(* IEC 61131-3 sources: cc_kush_rewrite/Functions/Bunker, 10 files *)

(* ---- FC_Bunker_CheckCriticalWeight.st ---- *)
FUNCTION FC_Bunker_CheckCriticalWeight : BOOL
VAR_INPUT
	Bunker1 : REFERENCE TO ST_Bunker;
	Bunker2 : REFERENCE TO ST_Bunker;
	Bunker3 : REFERENCE TO ST_Bunker;
END_VAR
VAR
END_VAR
// ========================================
// ПРОВЕРКА КРИТИЧЕСКИ НИЗКОГО ВЕСА
// ========================================
// Функция возвращает TRUE, если хотя бы один из бункеров достиг
// критически низкого уровня веса (сырье закончилось)
//
// ЛОГИКА:
// Когда определенное сырье заканчивается, вес бункера становится
// критически низким (rWeight <= BUNKER_WEIGHT_LIGHT_RED_SPECIAL).
// В этом случае необходимо подать красный сигнал на ВСЕ 3 бункера,
// чтобы прекратить подачу остального сырья. Далее они спокойно
// опустошаются в обычном автоматическом режиме.

FC_Bunker_CheckCriticalWeight :=
	(Bunker1.rWeight <= BUNKER_WEIGHT_LIGHT_RED_SPECIAL)
	OR (Bunker2.rWeight <= BUNKER_WEIGHT_LIGHT_RED_SPECIAL)
	OR (Bunker3.rWeight <= BUNKER_WEIGHT_LIGHT_RED_SPECIAL);

END_FUNCTION

(* ---- FC_Bunker_CheckEmptyBunker.st ---- *)
FUNCTION FC_Bunker_CheckEmptyBunker : BOOL
VAR_INPUT
	Bunker1 : REFERENCE TO ST_Bunker;
	Bunker2 : REFERENCE TO ST_Bunker;
	Bunker3 : REFERENCE TO ST_Bunker;
END_VAR
VAR
END_VAR
// ========================================
// ПРОВЕРКА ПОЛНОГО ОПУСТОШЕНИЯ БУНКЕРОВ
// ========================================
// Функция возвращает TRUE, если хотя бы один из бункеров полностью пуст.
//
// ЛОГИКА:
// Как только один из бункеров становится пустым (rWeight <= BUNKER_MINIMAL_WEIGHT),
// необходимо сразу остановить ВСЕ бункеры. Конвейер и отвалообразователь
// продолжают свою работу для транспортировки оставшегося материала.

FC_Bunker_CheckEmptyBunker :=
	(Bunker1.rWeight <= BUNKER_MINIMAL_WEIGHT)
	OR (Bunker2.rWeight <= BUNKER_MINIMAL_WEIGHT)
	OR (Bunker3.rWeight <= BUNKER_MINIMAL_WEIGHT);

END_FUNCTION

(* ---- FC_Bunker_CheckWeight.st ---- *)
FUNCTION FC_Bunker_CheckWeight : BOOL
VAR_INPUT
	Bunker : REFERENCE TO ST_Bunker;
END_VAR
VAR
END_VAR
// Проверка веса бункера. True - вес в порядке
FC_Bunker_CheckWeight := Bunker.rWeight > BUNKER_MINIMAL_WEIGHT;

END_FUNCTION

(* ---- FC_Bunker_EmergencyStop.st ---- *)
FUNCTION FC_Bunker_EmergencyStop : BOOL
VAR_INPUT
	Bunker : ST_Bunker;
END_VAR
VAR
	j : INT;
END_VAR
// Остановка моторов вибраторов (4 шт на бункер)
FOR j := 1 TO 4 DO
	Bunker.MotorVibrator[j].qxKM_Power := FALSE;
	Bunker.MotorVibrator[j].VFD.qxStart := FALSE;
	Bunker.MotorVibrator[j].VFD.Frequency.rTargetFrequency := 0.0;
	Bunker.MotorVibrator[j].VFD.qrOutFrequency := 0.0;
END_FOR

// Остановка моторов вибропитателей (2 шт на бункер)
FOR j := 1 TO 2 DO
	Bunker.MotorVibFeeder[j].qxKM_Power := FALSE;
	Bunker.MotorVibFeeder[j].VFD.qxStart := FALSE;
	Bunker.MotorVibFeeder[j].VFD.Frequency.rTargetFrequency := 0.0;
	Bunker.MotorVibFeeder[j].VFD.qrOutFrequency := 0.0;
END_FOR

// Установка красного сигнала светофора
FC_Bunker_SetLightColor(Bunker := Bunker, eColor := E_LightColor.RED);

END_FUNCTION

(* ---- FC_Bunker_GetErrorBunker.st ---- *)
FUNCTION FC_Bunker_GetErrorBunker : BOOL
VAR_INPUT
	Bunker : REFERENCE TO ST_Bunker;
END_VAR
VAR
END_VAR
FC_Bunker_GetErrorBunker :=
	FC_Bunker_GetErrorMotorVibFeeder(Bunker := Bunker)
	OR FC_Bunker_GetErrorMotorVibrator(motor := Bunker.MotorVibrator[1])
	OR FC_Bunker_GetErrorMotorVibrator(motor := Bunker.MotorVibrator[2])
	OR FC_Bunker_GetErrorMotorVibrator(motor := Bunker.MotorVibrator[3])
	OR FC_Bunker_GetErrorMotorVibrator(motor := Bunker.MotorVibrator[4]);

END_FUNCTION

(* ---- FC_Bunker_GetErrorMotorVibFeeder.st ---- *)
FUNCTION FC_Bunker_GetErrorMotorVibFeeder : BOOL
VAR_INPUT
	Bunker : REFERENCE TO ST_Bunker;
END_VAR
VAR
END_VAR
FC_Bunker_GetErrorMotorVibFeeder :=
		Bunker.MotorVibFeeder[1].VFD.fbStateFailure.qxInvertedSignal // Ошибка ЧРП (NC: TRUE=норма, инвертированный=TRUE=ошибка)
		OR Bunker.MotorVibFeeder[1].VFD.xStateFailureLocal // Ошибка ЧРП, полученная программным путём
		//OR Bunker.MotorVibFeeder[1].VFD.fbRangeDiagnostic.qxCriticalActive // Критическое значение тока эл. двигателя
		//OR NOT Bunker.MotorVibFeeder[1].fbStatorOverheat.qxSignal // Перегрев статора (1 - норма, 0 - перегрев)
		//OR Bunker.MotorVibFeeder[1].fbRangeDiagnostic[1].qxCriticalActive // Критический уровень нагрева подпишникового узла 1
		//OR Bunker.MotorVibFeeder[1].fbRangeDiagnostic[2].qxCriticalActive // Критический уровень нагрева подпишникового узла 2

		OR Bunker.MotorVibFeeder[2].VFD.fbStateFailure.qxInvertedSignal // Ошибка ЧРП (NC: TRUE=норма, инвертированный=TRUE=ошибка)
		OR Bunker.MotorVibFeeder[2].VFD.xStateFailureLocal; // Ошибка ЧРП, полученная программным путём
		//OR Bunker.MotorVibFeeder[2].VFD.fbRangeDiagnostic.qxCriticalActive // Критическое значение тока эл. двигателя
		//OR NOT Bunker.MotorVibFeeder[2].fbStatorOverheat.qxSignal // Перегрев статора (1 - норма, 0 - перегрев)
		//OR Bunker.MotorVibFeeder[2].fbRangeDiagnostic[1].qxCriticalActive // Критический уровень нагрева подпишникового узла 1
		//OR Bunker.MotorVibFeeder[2].fbRangeDiagnostic[2].qxCriticalActive; // Критический уровень нагрева подпишникового узла 2

END_FUNCTION

(* ---- FC_Bunker_GetErrorMotorVibrator.st ---- *)
FUNCTION FC_Bunker_GetErrorMotorVibrator : BOOL
VAR_INPUT
	motor : REFERENCE TO ST_Motor;
END_VAR
VAR
END_VAR
FC_Bunker_GetErrorMotorVibrator := (
	motor.VFD.fbStateFailure.qxInvertedSignal // Ошибка ЧРП (NC: TRUE=норма, инвертированный=TRUE=ошибка)
	OR motor.VFD.xStateFailureLocal // Ошибка ЧРП, полученная программным путём
	//OR motor.VFD.fbRangeDiagnostic.qxCriticalActive // Критическое значение тока эл. двигателя
);

END_FUNCTION

(* ---- FC_Bunker_GetErrorWeight.st ---- *)
FUNCTION FC_Bunker_GetErrorWeight : BOOL
VAR_INPUT
	Bunker1 : REFERENCE TO ST_Bunker;
	Bunker2 : REFERENCE TO ST_Bunker;
	Bunker3 : REFERENCE TO ST_Bunker;
END_VAR
VAR
END_VAR
// Если 2 или больше бункеров являются пустыми, мы получаем ошибку
FC_Bunker_GetErrorWeight :=
	2 > BOOL_TO_INT(FC_Bunker_CheckWeight(Bunker := Bunker1))
	  + BOOL_TO_INT(FC_Bunker_CheckWeight(Bunker := Bunker2))
	  + BOOL_TO_INT(FC_Bunker_CheckWeight(Bunker := Bunker3));

END_FUNCTION

(* ---- FC_Bunker_GetLightColor.st ---- *)
FUNCTION FC_Bunker_GetLightColor : E_LightColor
VAR_INPUT
	irWeight : REAL; // Вес текущего бункера
	xCriticalWeightDetected : BOOL; // Глобальный флаг критического веса (хотя бы один бункер достиг критической уставки)
	xThisBunkerIsCritical : BOOL; // Флаг того, что ЭТОТ конкретный бункер находится в критическом состоянии
	xBunkerWorking : BOOL; // Бункер работает (питатели активны)
END_VAR
VAR
END_VAR

// ========================================
// ПРИОРИТЕТНАЯ ПРОВЕРКА: КРИТИЧЕСКИЙ ВЕС
// ========================================
// ЛОГИКА:
// 1. Если хотя бы один бункер достиг критически низкого веса (сырье закончилось),
//    то ЭТОТ конкретный бункер горит ЗЕЛЁНЫМ (приоритет на заполнение),
//    а ВСЕ ОСТАЛЬНЫЕ бункеры горят КРАСНЫМ (остановить заполнение).
// 2. Как только критический бункер выходит на норму (вес >= BUNKER_WEIGHT_LIGHT_GREEN),
//    система возвращается к обычному режиму работы светофоров.

IF xCriticalWeightDetected THEN
	// Если этот конкретный бункер находится в критическом состоянии
	IF xThisBunkerIsCritical THEN
		// Этот бункер горит ЗЕЛЁНЫМ (срочно заполнить!)
		FC_Bunker_GetLightColor := E_LightColor.GREEN;
	ELSE
		// Все остальные бункеры горят КРАСНЫМ (прекратить заполнение!)
		FC_Bunker_GetLightColor := E_LightColor.RED;
	END_IF;
	RETURN;
END_IF;

// ========================================
// ОБЫЧНАЯ РАБОТА: ОПРЕДЕЛЕНИЕ ЦВЕТА ПО ВЕСУ
// ========================================
IF irWeight >= BUNKER_WEIGHT_LIGHT_RED THEN
	// Вес выше или равен уставке RED - красный сигнал (бункер полный, прекратить загрузку)
	FC_Bunker_GetLightColor := E_LightColor.RED;

ELSIF irWeight >= BUNKER_WEIGHT_LIGHT_YELLOW THEN
	// Вес между YELLOW и RED - жёлтый сигнал (бункер заполнен умеренно)
	FC_Bunker_GetLightColor := E_LightColor.YELLOW;

ELSIF irWeight >= BUNKER_WEIGHT_LIGHT_GREEN THEN
	// Вес между GREEN и YELLOW - зелёный сигнал (можно загружать)
	FC_Bunker_GetLightColor := E_LightColor.GREEN;

ELSE
	// Вес ниже GREEN - выключен (недостаточный вес для работы)
	// Если бункер работает, оставляем зелёный, иначе - выключен
	IF xBunkerWorking THEN
		FC_Bunker_GetLightColor := E_LightColor.GREEN;
	ELSE
		FC_Bunker_GetLightColor := E_LightColor.OFF;
	END_IF;
END_IF;

END_FUNCTION

(* ---- FC_Bunker_SetLightColor.st ---- *)
FUNCTION FC_Bunker_SetLightColor : BOOL
VAR_INPUT
	Bunker : REFERENCE TO ST_Bunker;
	eColor : E_LightColor;
END_VAR
VAR
END_VAR
// Сброс всех сигналов
Bunker.qxLightRed := FALSE;
Bunker.qxLightYellow := FALSE;
Bunker.qxLightGreen := FALSE;

// Установка нужного цвета
CASE eColor OF
	E_LightColor.RED:
		Bunker.qxLightRed := TRUE;
		Bunker.eLightColor := E_LightColor.RED;

	E_LightColor.YELLOW:
		Bunker.qxLightYellow := TRUE;
		Bunker.eLightColor := E_LightColor.YELLOW;

	E_LightColor.GREEN:
		Bunker.qxLightGreen := TRUE;
		Bunker.eLightColor := E_LightColor.GREEN;

	E_LightColor.OFF:
		// Все уже выключены
		Bunker.eLightColor := E_LightColor.OFF;
END_CASE;

FC_Bunker_SetLightColor := TRUE;

END_FUNCTION
